// TIA Portal V16 export
// export: Created 2022-02-28T20:45:45.477533Z, ExportSetting WithDefaults, DisplayName Totally Integrated Automation Portal, DisplayVersion V16, DisplayName TIA Portal Version Control Interface, DisplayVersion V16, DisplayName TIA Portal Openness, DisplayVersion V16, DisplayName STEP 7 Professional, DisplayVersion V16, DisplayName STEP 7 Safety, DisplayVersion V16, DisplayName WinCC Advanced, DisplayVersion V16
FUNCTION_BLOCK "DataMan"   // FB1, LAD
TITLE = Cámara Cognex DataMan
{ S7_Optimized_Access := 'TRUE' }
VERSION : 0.1
// stored: AutoNumber true, IsIECCheckEnabled false, IsRetainMemResEnabled false, MemoryReserve 100, SetENOAutomatically false, UDAEnableTagReadback false
   VAR_OUTPUT
      DataMan_Trigger_Ready : Bool;
      DataMan_TriggerAck : Bool;
      DataMan_ResultAvailable : Bool;
      DataMan_ResultID : Word;
      "DataMan Result Code" : Word;
      "DataMan Result Length" : Word;
      ResultData : Array[0..63] of Byte;
   END_VAR
   VAR_IN_OUT
      DataMan_Trigger_Enable : Bool;
      DataMan_Trigger : Bool;
      DataMan_ResultsAck : Bool;
   END_VAR
   VAR
      Resultado_Pendiente : Bool;
      "Lastest Result" : Struct
         ID : Int;
         Flags : Int;
         Lenght : Int;
         Value : Array[0..63] of Byte;
      END_STRUCT;
   END_VAR
   VAR_TEMP   // added for the SCL form of the ladder/FBD networks
      _w1 : Bool;
   END_VAR
BEGIN

REGION Network 1: Habilitar Comunicación Profinet
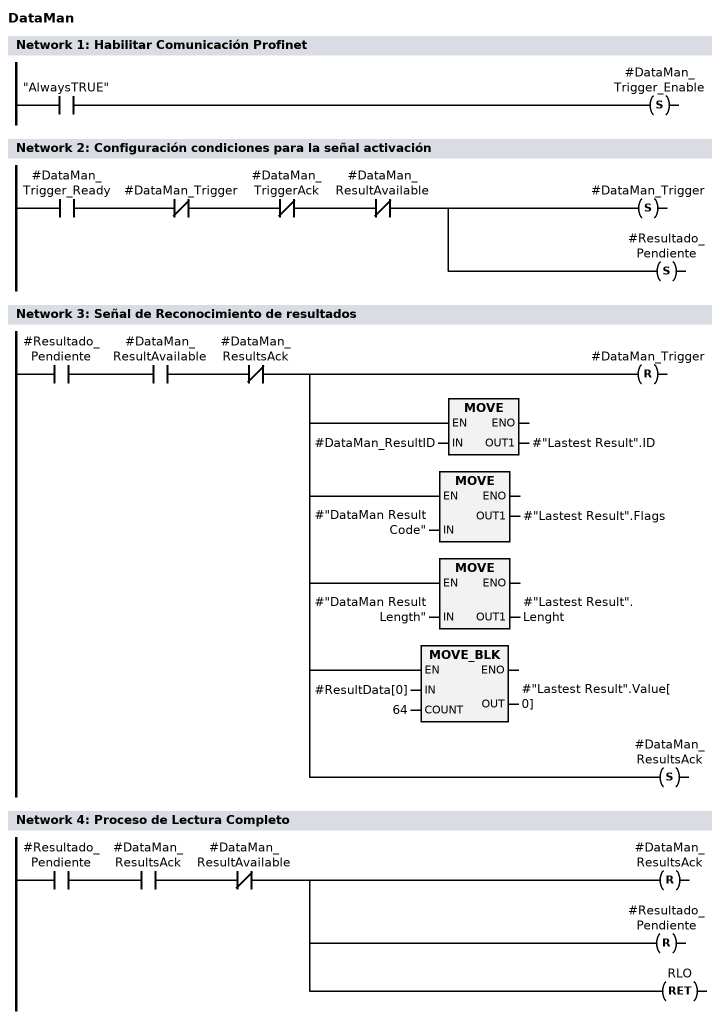
   RUNG wire#powerrail
      Contact( "AlwaysTRUE" )
      S_Coil( #DataMan_Trigger_Enable )
   END_RUNG
   // the same network as SCL:
   IF "AlwaysTRUE" THEN #DataMan_Trigger_Enable := TRUE; END_IF;
END_REGION

REGION Network 2: Configuración condiciones para la señal activación
   RUNG wire#powerrail
      Contact( #DataMan_Trigger_Ready )
      I_Contact( #DataMan_Trigger )
      I_Contact( #DataMan_TriggerAck )
      I_Contact( #DataMan_ResultAvailable )
      wire#w1
      S_Coil( #DataMan_Trigger )
   END_RUNG
   RUNG wire#w1
      S_Coil( #Resultado_Pendiente )
   END_RUNG
   // the same network as SCL:
   #_w1 := #DataMan_Trigger_Ready AND NOT #DataMan_Trigger AND NOT #DataMan_TriggerAck AND NOT #DataMan_ResultAvailable;
   IF #_w1 THEN
       #DataMan_Trigger := TRUE;
       #Resultado_Pendiente := TRUE;
   END_IF;
END_REGION

REGION Network 3: Señal de Reconocimiento de resultados
   IF #Resultado_Pendiente AND #DataMan_ResultAvailable AND NOT #DataMan_ResultsAck THEN
       #DataMan_Trigger := FALSE;
       #"Lastest Result".ID := #DataMan_ResultID;
       #"Lastest Result".Flags := #"DataMan Result Code";
       #"Lastest Result".Lenght := #"DataMan Result Length";
       MOVE_BLK(IN := #ResultData[0], COUNT := 64, OUT => #"Lastest Result".Value[0]);
       #DataMan_ResultsAck := TRUE;
   END_IF;
END_REGION

REGION Network 4: Proceso de Lectura Completo
   #_w1 := #Resultado_Pendiente AND #DataMan_ResultsAck AND NOT #DataMan_ResultAvailable;
   IF #_w1 THEN
       #DataMan_ResultsAck := FALSE;
       #Resultado_Pendiente := FALSE;
       ENO := TRUE;
       RETURN;
   END_IF;
END_REGION
END_FUNCTION_BLOCK
